(* IEC 61131-3 sources: repolevel_ST_code_completion/dataset/project_code/轴控/FB105_轴控制集/FB51_调模A轴控制, 4 files *)

(* ---- A01_轴控主块.st ---- *)
PROGRAM A01_轴控主块
VAR
    FB_AxisControl_调模A轴 : FB_轴控块; (* 声明位置设置功能块 *)
    FB_AxisStop_调模A轴 : FB_轴停止触发块;
    SMC_ChangeGearingRatio0 : SMC_ChangeGearingRatio;
    SMC_SetControllerMode0 : SMC_SetControllerMode;
    SMC_SetTorque0 : SMC_SetTorque;
    bDone_SetMode : BOOL;
END_VAR

VAR_INPUT
END_VAR

VAR_OUTPUT
END_VAR

VAR_IN_OUT
END_VAR

FB_AxisControl_调模A轴(
    Enable := , // 使能轴（可根据实际逻辑控制）
    JogFor := b调模A轴正向点动,
    JogBack := b调模A轴反向点动,
    JogVelocity := r调模A轴点动速度给定,
    StopExcute := b调模A轴停止触发,
    ResetExcute := HMI_b复位,
    AbsExcute := , // 初始设为FALSE，需触发时置TRUE
    AbsPosition := r调模A轴绝对运动位置给定,
    AbsVelocity := r调模A轴绝对运动速度给定,
    // AbsAcceleration 等参数若有默认值或无需外部给定，可省略或按实际赋值
    AbsAcceleration := ,
    AbsDeceleration := ,
    RelExcute := ,
    RelPosition := r调模A轴相对运动位置给定,
    RelVelocity := r调模A轴相对运动速度给定,
    // RelAcceleration 等参数同理
    RelAcceleration := ,
    RelDeceleration := ,
    VelExcute := ,
    VelVelocity := r调模A轴速度模式速度给定,
    InchForward := ,
    InchBackward := ,
    InchDistance := r调模A轴寸动位置给定,
    InchVelocity := r调模A轴寸动速度给定,
    // InchAcceleration 等参数同理
    InchAcceleration := ,
    InchDeceleration := ,
    SetPosExcute := ,
    ReStartSlaveEx := ,
    AxisName := AxisLeftTiaoMo,

    // 输出映射
    EnableStatus => b调模A轴使能OK,
    StopDone => b调模A轴停止完成,
    AbsDone => b调模A轴绝对运动完成,
    RelDone => b调模A轴相对运动完成,
    VelBusy => b调模A轴速度模式Busy,
    InchBusy => b调模A轴寸动模式Busy,
    AxisStandsstill => b调模A轴停止中,
    AbsBusy => b调模A轴绝对模式Busy,
    RelBusy => b调模A轴相对模式Busy,
    AxisError => b调模A轴错误,
    AxisAccing => b调模A轴加速中,
    AxisDecing => b调模A轴减速中,
    FBErrorOccured => ,
    Homing => ,
    Stopping => ,
    ErrorID => ,
    SetPosDone => ,
    bOperational => ,
    eComState => ,
    wComState => ,
    JogBusy => b调模A轴点动模式Busy
    ReStartSlaveDone =>
    // 其他输出需按功能块定义补充映射
);

FB_AxisStop_调模A轴(
    StopExcute := b调模A轴停止触发
);

SMC_ClearFBError_Instance(
    EN := FBErrorOccurred,
    pDrive := ADR(AxisLeftTiaoMo),
    ENO => ,
    SMC_ClearFBError =>
);

SMC_ChangeGearingRatio0(
    Axis := AxisLeftTiaoMo,
    bExecute := ,
    dwRatioTechUnitsDenom := AxisLeftTiaoMo.dwRatioTechUnitsDenom,
    iRatioTechUnitsNum := REAL_TO_INT(HMI_r调模A轴导程),
    fPositionPeriod := fPositionPeriod,
    iMovementType := SMC_MOVEMENTTYPE.linear,

    bDone => ,
    bBusy => ,
    bError => ,
    nErrorID =>
);

AxisLeftTiaoMo_iRestNumerator := 0;

SMC_SetControllerMode0(
    Axis := AxisLeftTiaoMo,
    bExecute := ,
    nControllerMode := SMC_CONTROLLER_MODE.SMC_torque,
    bDone => bDone_SetMode,
    bBusy => ,
    bError => ,
    nErrorID =>
);

// 调用 SMC_SetTorque 功能块，设置扭矩
SMC_SetTorque0(
    Axis := AxisLeftTiaoMo,
    bEnable := bDone_SetMode,
    fTorque := ,
    bBusy => ,
    bError => ,
    nErrorID =>
);

(* ---- A02_数据运算.st ---- *)
(*基本速度，位置*)
r调模A轴点动速度给定:=HMI_r调模A轴手动速度;

r调模A轴绝对运动速度给定:=HMI_r调模A轴自动速度;
r调模A轴相对运动速度给定:=HMI_r调模A轴自动速度;
r调模A轴速度模式速度给定:=HMI_r调模A轴自动速度;
r调模A轴寸动速度给定:=HMI_r调模A轴自动速度;

HMI_r调模A轴当前位置:=LREAL_TO_REAL(AxisLeftTiaoMo.fActPosition);
HMI_r调模A轴当前速度:=LREAL_TO_REAL(AxisLeftTiaoMo.fActVelocity);

FB_AxisControl_调模A轴.AbsAcceleration:=r调模A轴绝对运动速度给定/(HMI_r调模A轴加速时间/1000);
FB_AxisControl_调模A轴.AbsDeceleration:=r调模A轴绝对运动速度给定/(HMI_r调模A轴减速时间/1000);

FB_AxisControl_调模A轴.RelAcceleration:=r调模A轴相对运动速度给定/(HMI_r调模A轴加速时间/1000);
FB_AxisControl_调模A轴.RelDeceleration:=r调模A轴相对运动速度给定/(HMI_r调模A轴减速时间/1000);

FB_AxisControl_调模A轴.InchAcceleration:=r调模A轴寸动速度给定/(HMI_r调模A轴加速时间/1000);
FB_AxisControl_调模A轴.InchDeceleration:=r调模A轴寸动速度给定/(HMI_r调模A轴减速时间/1000);

(*正负限位*)
IF b调模A轴启用限位 AND b调模A轴回零完成 THEN
	AxisLeftTiaoMo.bSWLimitEnable:=TRUE;
	AxisLeftTiaoMo.fSWLimitPositive:=HMI_r调模A轴正限位;
	AxisLeftTiaoMo.fSWLimitNegative:=HMI_r调模A轴负限位;
	AxisLeftTiaoMo.fSWLimitDeceleration:=1000000;
	ELSE
	AxisLeftTiaoMo.bSWLimitEnable:=FALSE;
END_IF

(* ---- A03_原点回归.st ---- *)
PROGRAM A03_原点回归
VAR
    MC_SetPosition_0 : SM3_Basic.MC_SetPosition; (* 声明位置设置功能块 *)
    SMC_Homing_0 : SM3_Basic.SMC_Homing;
END_VAR

VAR_INPUT
END_VAR

VAR_OUTPUT
END_VAR

VAR_IN_OUT
END_VAR

(* 调用MC_SetPosition功能块，实现轴位置设置 *)
MC_SetPosition_0(
    Axis := AxisLeftTiaoMo,
    Execute := ,
    Position := 0,
    Mode := 0,
    Done => ,
    Busy => ,
    Error => ,
    ErrorID =>
);

SMC_Homing_0(
    Axis := AxisLeftTiaoMo,
    bExecute := ,
    fHomePosition := 0,
    fVelocitySlow := HMI_r调模A轴回零慢速,
    fVelocityFast := HMI_r调模A轴回零快速,
    fAcceleration := HMI_r调模A轴回零快速*10000,
    fDeceleration := HMI_r调模A轴回零快速*10000,
    fJerk := ,
    nDirection := -1,
    bReferenceSwitch := DI_调模A步进原点,
    fSignalDelay := ,
    nHomingMode := 1,
    bReturnToZero := ,
    bIndexOccured := ,
    fIndexPosition := ,
    bIgnoreHWLimit := ,
    bDone => ,
    bBusy => ,
    bCommandAborted => ,
    bError => ,
    nErrorID => ,
    bStartLatchingIndex =>
);

(* ---- FB51_调模A轴控制.st ---- *)
PROGRAM FB51_调模A轴控制
VAR
	FB_AxisMotionDiag_调模A轴: FB_轴通讯状态块;
	FB_AxisStop_调模A轴: FB_轴停止触发块;

	SMC_SetControllerMode0: SMC_SetControllerMode;
	SMC_SetTorque0: SMC_SetTorque;
	SMC_ChangeGearingRatio0: SMC_ChangeGearingRatio;
    MC_SetPosition_0: SM3_Basic.MC_SetPosition;
	SMC_Homing_0: SM3_Basic.SMC_Homing;

	fb_CommunicationOK: TON;

	R_TRIG回零: R_TRIG;
	R_TRIG初始化回零: R_TRIG;
	b调模A轴手动定位: BOOL;
END_VAR

(*轴通讯状态*)
b调模A轴通讯OK:=FB_AxisMotionDiag_调模A轴.EtherCATBusOK;

FB_AxisMotionDiag_调模A轴(Axis_bCommunication:= AxisLeftTiaoMo.bCommunication,
                        Axis_wCommunicationState:= AxisLeftTiaoMo.wCommunicationState,
                        EtherCATBusOK=> );

fb_CommunicationOK(IN:= b调模A轴通讯OK, PT:= T#3S, Q=> , ET=> );

(*轴使能操作*)
IF NOT HMI_b调模A轴断使能 AND fb_CommunicationOK.Q THEN
	FB_AxisControl_调模A轴.Enable:=TRUE;
	ELSE
	FB_AxisControl_调模A轴.Enable:=FALSE;
END_IF

(*轴控点动*)
IF HMI_b调模A轴正向点动 AND b调模A轴使能OK AND NOT b调模A轴错误 AND b非急停手动模式 AND NOT b调模A轴反向点动 THEN
	b调模A轴正向点动:=TRUE;
	ELSE
	b调模A轴正向点动:=FALSE;
END_IF
IF HMI_b调模A轴反向点动 AND b调模A轴使能OK AND NOT b调模A轴错误 AND b非急停手动模式 AND NOT b调模A轴正向点动 THEN
	b调模A轴反向点动:=TRUE;
	ELSE
	b调模A轴反向点动:=FALSE;
END_IF

(*轴控寸动*)
IF b调模A轴正向寸动 AND b调模A轴使能OK AND NOT b调模A轴错误 AND NOT FB_AxisControl_调模A轴.InchBackward THEN
	FB_AxisControl_调模A轴.InchForward:=TRUE;
	ELSE
	FB_AxisControl_调模A轴.InchForward:=FALSE;
END_IF
IF b调模A轴反向寸动 AND b调模A轴使能OK AND NOT b调模A轴错误 AND NOT FB_AxisControl_调模A轴.InchForward THEN
	FB_AxisControl_调模A轴.InchBackward:=TRUE;
	ELSE
	FB_AxisControl_调模A轴.InchBackward:=FALSE;
END_IF

(*轴控回零*)
R_TRIG回零(CLK:= SMC_Homing_0.bDone, Q=> );
R_TRIG初始化回零(CLK:= b调模A轴回零触发, Q=> );
IF (HMI_b调模A轴单独回原 OR R_TRIG初始化回零.Q) AND b调模A轴使能OK AND NOT b调模A轴错误 AND b非急停手动模式 AND NOT SMC_Homing_0.bBusy THEN
	SMC_Homing_0.bExecute:=TRUE;
END_IF
IF R_TRIG回零.Q THEN
	b调模A轴回零完成:=TRUE;
	SMC_Homing_0.bExecute:=FALSE;
END_IF

(*轴控绝对运动*)
IF b调模A轴绝对运动触发 AND b调模A轴使能OK AND NOT b调模A轴错误 THEN
	FB_AxisControl_调模A轴.AbsExcute:=TRUE;
	ELSE
	FB_AxisControl_调模A轴.AbsExcute:=FALSE;
END_IF

(*轴控相对运动*)
IF b调模A轴相对运动触发 AND b调模A轴使能OK AND NOT b调模A轴错误 THEN
	FB_AxisControl_调模A轴.RelExcute:=TRUE;
	ELSE
	FB_AxisControl_调模A轴.RelExcute:=FALSE;
END_IF

(*轴控定位*)
IF HMI_b调模A轴去工作位 AND b调模A轴使能OK AND NOT b调模A轴错误 AND b非急停手动模式 AND NOT b调模A轴绝对模式Busy AND NOT b调模A轴手动定位 THEN
	r调模A轴绝对运动位置给定:=HMI_r调模A轴宽度位置;
	b调模A轴绝对运动触发:=TRUE;
	b调模A轴手动定位:=TRUE;
END_IF
IF b调模A轴手动定位 AND b调模A轴绝对运动触发 AND b调模A轴绝对运动完成 THEN
	b调模A轴绝对运动触发:=FALSE;
	b调模A轴手动定位:=FALSE;
END_IF
